TYPE Application :
STRUCT
	GearingType			:	GearingType;
END_STRUCT
END_TYPE

(* stored: Version 1.1.0.1, ProductVersion 3.1.4024.6
   DUT Application: Id {b8ff7bc1-c45a-4a5f-91e6-692a392be699} *)
